(* IEC 61131-3 sources: ScaleLib/, 6 files *)

(* ---- ScaleLib.typ ---- *)
(********************************************************************
 * COPYRIGHT --
 ********************************************************************
 * Library: Scale_Lib
 * File: Scale_Lib.typ
 * Author: David
 * Created: August 10, 2010
 ********************************************************************
 * Data types of library Scale_Lib
 ********************************************************************)

TYPE
	Scale_OUT_STAT_typ : 	STRUCT
		Error : BOOL;
	END_STRUCT;
	Scale_OUT_typ : 	STRUCT
		OutputValue : REAL;
		STAT : Scale_OUT_STAT_typ;
	END_STRUCT;
	Scale_IN_CFG_Point_typ : 	STRUCT
		Input : REAL;
		Output : REAL;
	END_STRUCT;
	Scale_IN_CFG_typ : 	STRUCT
		Point : ARRAY[0..1] OF Scale_IN_CFG_Point_typ;
	END_STRUCT;
	Scale_IN_typ : 	STRUCT
		InputValue : REAL;
		CFG : Scale_IN_CFG_typ;
	END_STRUCT;
	Scale_typ : 	STRUCT
		IN : Scale_IN_typ;
		OUT : Scale_OUT_typ;
	END_STRUCT;
END_TYPE

(* ---- C_to_F.st ---- *)
(********************************************************************
 * COPYRIGHT --
 ********************************************************************
 * Library: Scale_Lib
 * File: C_to_F.st
 * Author: David
 * Created: September 10, 2010
 ********************************************************************
 * Implementation of library Scale_Lib
 ********************************************************************)

(********************************************************************)
(* Converts from degrees Celsius to degrees Fahrenheit 				*)
(********************************************************************)

(* DONE and TESTED DFB *)

FUNCTION C_to_F

C_to_F:=  C * 1.8 + 32.0;

END_FUNCTION

(* ---- F_to_C.st ---- *)
(********************************************************************
 * COPYRIGHT --
 ********************************************************************
 * Library: Scale_Lib
 * File: F_to_C.st
 * Author: David
 * Created: September 10, 2010
 ********************************************************************
 * Implementation of library Scale_Lib
 ********************************************************************)

(********************************************************************)
(* Converts from degrees Fahrenheit to degrees Celsius 				*)
(********************************************************************)

(* DONE and TESTED DFB *)

FUNCTION F_to_C

F_to_C:=  ( F - 32.0 ) / 1.8;

END_FUNCTION

(* ---- ScaleFnCyclic.st ---- *)
(********************************************************************
 * COPYRIGHT --
 ********************************************************************
 * Library: Scale_Lib
 * File: ScaleFnCyclic.st
 * Author: David
 * Created: July 21, 2010
 ********************************************************************
 * Implementation of library Scale_Lib
 ********************************************************************)

(****************************************************************************************)
(* Cyclic function for scaling 															*)
(****************************************************************************************)

(* Error checking			DONE and TESTED DFB 20110512 *)
(* Scaling					DONE and TESTED DFB 20110512 *)

FUNCTION ScaleFnCyclic

(************************************************************)
(* Set return value to get rid of compile warning 			*)
(************************************************************)

ScaleFnCyclic:=	FALSE;

(************************************************************)
(* Check for errors and scale values			 			*)
(************************************************************)

IF( (t.IN.CFG.Point[0].Input = t.IN.CFG.Point[1].Input) )THEN

	t.OUT.OutputValue:=	0;
	t.OUT.STAT.Error:=	1;

ELSE

	t.OUT.OutputValue:= 	t.IN.CFG.Point[0].Output +
							( ( t.IN.CFG.Point[1].Output - t.IN.CFG.Point[0].Output ) / (t.IN.CFG.Point[1].Input - t.IN.CFG.Point[0].Input) ) *
							( t.IN.InputValue - t.IN.CFG.Point[0].Input );

	t.OUT.STAT.Error:=	0;

END_IF

END_FUNCTION

(* ---- ScaleLib.fun ---- *)
(********************************************************************
 * COPYRIGHT --
 ********************************************************************
 * Library: Scale_Lib
 * File: Scale_Lib.fun
 * Author: David
 * Created: August 10, 2010
 ********************************************************************
 * Functions and function blocks of library Scale_Lib
 ********************************************************************)

FUNCTION ScaleFnCyclic : BOOL (*Cyclic function for scaling*)
	VAR_IN_OUT
		t : Scale_typ; (*Scale control object*)
	END_VAR
END_FUNCTION

FUNCTION F_to_C : REAL (*Converts from degrees Fahrenheit to degrees Celsius*)
	VAR_INPUT
		F : REAL; (*Temperature in degrees Fahrenheit*)
	END_VAR
END_FUNCTION

FUNCTION C_to_F : REAL (*Converts from degrees Celsius to degrees Fahrenheit*)
	VAR_INPUT
		C : REAL; (*Temperature in degrees Celsius*)
	END_VAR
END_FUNCTION

(* ---- ScaleLib.var ---- *)
(********************************************************************
 * COPYRIGHT --
 ********************************************************************
 * Library: Scale_Lib
 * File: Scale_Lib.var
 * Author: David
 * Created: August 10, 2010
 ********************************************************************
 * Constants of library Scale_Lib
 ********************************************************************)

VAR CONSTANT

END_VAR
